{attribute addProperty BoxType "EP1312-0001-0016"}
{attribute addProperty Id "InfoDataInfoData_192954DE162"}
{attribute addProperty CRC "395970889"}
{attribute addProperty SizeInBites "16"}
{attribute addProperty SizeInBytes "2"}
TYPE EP1312_179A0949 :
STRUCT
	{attribute addProperty Name "InfoData"}
	InfoData : InfoData_192954DE;
END_STRUCT
END_TYPE

(* stored: Version 1.2.0.0, ProductVersion 3.1.4024.9
   DUT EP1312_179A0949: Id {0c54a1e0-f83f-47b0-82d9-8e123d82598b} *)
